{attribute 'GeneratedUsingTerminal: EPP9001-0060-0016'}
{attribute addProperty BoxType "EPP9001-0060-0016"}
{attribute addProperty Id "EtcSlaveTerminalBaseInfoDataAT %I*InfoData_6F19DB2B2"}
{attribute addProperty CRC "2874840167"}
{attribute addProperty Size "2"}
TYPE EPP9001_AB5A9467 EXTENDS EtcSlaveTerminalBase :
STRUCT
	{attribute addProperty Name "InfoData"}
	InfoData : InfoData_6F19DB2B;
END_STRUCT
END_TYPE

(* stored: Version 1.2.0.0, ProductVersion 3.1.4024.9
   DUT EPP9001_AB5A9467: Id {20eb080a-6505-4d60-a35d-ee6156a0b904} *)
